COMM ARCOF
COMM SMOVL C00540 BC00540 V=400.0  +MOVJ EC00540
COMM SMOVL C00541 BC00541 V=1000.0  +MOVJ EC00541
COMM SFTOF3D
'Path W1887
SFTOF3D
SFTON3D P023
MOVJ C00542 BC00542 VJ=100.00  +MOVJ EC00542 VJ=100.00
SMOVL C00543 BC00543 V=400.0  +MOVJ EC00543
SMOVL C00544 BC00544 V=100.0 PL=0  +MOVJ EC00544
SREFP 1 C00545 BC00545  +REFP EC00545
SREFP 2 C00546 BC00546  +REFP EC00546
MACRO1 MJ#(0) ARGF9
ARCON
SMOVL C00547 BC00547 V=10.0  +MOVJ EC00547
ARCOF
SMOVL C00548 BC00548 V=400.0  +MOVJ EC00548
SMOVL C00549 BC00549 V=1000.0  +MOVJ EC00549
SFTOF3D
MOVJ C00550 BC00550 VJ=100.00  +MOVJ EC00550 VJ=100.00
MOVJ C00551 BC00551 VJ=100.00  +MOVJ EC00551 VJ=100.00
MOVJ C00552 BC00552 VJ=100.00  +MOVJ EC00552 VJ=100.00
'2
MOVJ C00553 BC00553 VJ=100.00  +MOVJ EC00553 VJ=100.00
MOVJ C00554 BC00554 VJ=100.00  +MOVJ EC00554 VJ=20.00
MOVJ C00555 BC00555 VJ=100.00  +MOVJ EC00555 VJ=100.00
'Path W1888
SFTOF3D
SFTON3D P021
MOVJ C00556 BC00556 VJ=15.00  +MOVJ EC00556 VJ=100.00
SMOVL C00557 BC00557 V=400.0  +MOVJ EC00557
SMOVL C00558 BC00558 V=133.3 PL=0  +MOVJ EC00558
SREFP 1 C00559 BC00559  +REFP EC00559
SREFP 2 C00560 BC00560  +REFP EC00560
MACRO1 MJ#(0) ARGF14
ARCON
SMOVL C00561 BC00561 V=10.0  +MOVJ EC00561
ARCOF
SMOVL C00562 BC00562 V=166.7  +MOVJ EC00562
SMOVL C00563 BC00563 V=166.7  +MOVJ EC00563
MACRO1 MJ#(0) ARGF14
SMOVL C00564 BC00564 V=133.3 PL=0  +MOVJ EC00564
ARCON
SMOVL C00565 BC00565 V=10.0  +MOVJ EC00565
ARCOF
SMOVL C00566 BC00566 V=400.0  +MOVJ EC00566
SFTOF3D
MOVJ C00567 BC00567 VJ=50.00  +MOVJ EC00567 VJ=20.00
MOVJ C00568 BC00568 VJ=100.00  +MOVJ EC00568 VJ=100.00
'Path W1889
SFTOF3D
SFTON3D P021
MOVJ C00569 BC00569 VJ=100.00  +MOVJ EC00569 VJ=100.00
MOVJ C00570 BC00570 VJ=100.00  +MOVJ EC00570 VJ=100.00
SMOVL C00571 BC00571 V=400.0  +MOVJ EC00571
SMOVL C00572 BC00572 V=133.3 PL=0  +MOVJ EC00572
SREFP 1 C00573 BC00573  +REFP EC00573
SREFP 2 C00574 BC00574  +REFP EC00574
MACRO1 MJ#(0) ARGF14
ARCON
SMOVL C00575 BC00575 V=10.0  +MOVJ EC00575
ARCOF
SMOVL C00576 BC00576 V=166.7  +MOVJ EC00576
SMOVL C00577 BC00577 V=166.7  +MOVJ EC00577
SMOVL C00578 BC00578 V=166.7 PL=0  +MOVJ EC00578
ARCON
SMOVL C00579 BC00579 V=10.0  +MOVJ EC00579
ARCOF
SMOVL C00580 BC00580 V=400.0  +MOVJ EC00580
SMOVL C00581 BC00581 V=1000.0  +MOVJ EC00581
SMOVL C00582 BC00582 V=1000.0  +MOVJ EC00582
SFTOF3D
MOVJ C00583 BC00583 VJ=100.00  +MOVJ EC00583 VJ=20.00
MOVJ C00584 BC00584 VJ=100.00  +MOVJ EC00584 VJ=100.00
MOVJ C00585 BC00585 VJ=100.00  +MOVJ EC00585 VJ=100.00
MOVJ C00586 BC00586 VJ=100.00  +MOVJ EC00586 VJ=100.00
MOVJ C00587 BC00587 VJ=100.00  +MOVJ EC00587 VJ=100.00
'3
'Path W1890
SFTOF3D
SFTON3D P023
MOVJ C00588 BC00588 VJ=100.00  +MOVJ EC00588 VJ=100.00
'BRAKUJACY ELEMENT
COMM SMOVL C00589 BC00589 V=400.0  +MOVJ EC00589
COMM SMOVL C00590 BC00590 V=100.0 PL=0  +MOVJ EC00590
COMM SREFP 1 C00591 BC00591  +REFP EC00591
COMM SREFP 2 C00592 BC00592  +REFP EC00592
COMM MACRO1 MJ#(0) ARGF0
COMM ARCON
COMM SMOVL C00593 BC00593 V=10.0  +MOVJ EC00593
COMM SMOVL C00594 BC00594 V=10.0  +MOVJ EC00594
COMM SMOVL C00595 BC00595 V=10.0  +MOVJ EC00595
COMM ARCOF
COMM SMOVL C00596 BC00596 V=400.0  +MOVJ EC00596
COMM SMOVL C00597 BC00597 V=1000.0  +MOVJ EC00597
SFTOF3D
'Path W1891
SFTOF3D
SFTON3D P023
MOVJ C00598 BC00598 VJ=100.00  +MOVJ EC00598 VJ=100.00
SMOVL C00599 BC00599 V=400.0  +MOVJ EC00599
SMOVL C00600 BC00600 V=133.3 PL=0  +MOVJ EC00600
SREFP 1 C00601 BC00601  +REFP EC00601
SREFP 2 C00602 BC00602  +REFP EC00602
MACRO1 MJ#(0) ARGF14
ARCON
SMOVL C00603 BC00603 V=11.7  +MOVJ EC00603
ARCOF
SMOVL C00604 BC00604 V=400.0  +MOVJ EC00604
SMOVL C00605 BC00605 V=1000.0  +MOVJ EC00605
SFTOF3D
MOVJ C00606 BC00606 VJ=100.00  +MOVJ EC00606 VJ=100.00
MOVJ C00607 BC00607 VJ=100.00  +MOVJ EC00607 VJ=20.00
MOVJ C00608 BC00608 VJ=100.00  +MOVJ EC00608 VJ=100.00
MOVJ C00609 BC00609 VJ=100.00  +MOVJ EC00609 VJ=20.00
MOVJ C00610 BC00610 VJ=100.00  +MOVJ EC00610 VJ=100.00
MOVJ C00611 BC00611 VJ=100.00  +MOVJ EC00611 VJ=100.00
'4
'Path W1892
SFTOF3D
SFTON3D P022
MOVJ C00612 BC00612 VJ=100.00  +MOVJ EC00612 VJ=20.00
SMOVL C00613 BC00613 V=400.0  +MOVJ EC00613
SMOVL C00614 BC00614 V=133.3 PL=0  +MOVJ EC00614
SREFP 1 C00615 BC00615  +REFP EC00615
SREFP 2 C00616 BC00616  +REFP EC00616
MACRO1 MJ#(0) ARGF14
ARCON
SMOVL C00617 BC00617 V=10.0  +MOVJ EC00617
ARCOF
SMOVL C00618 BC00618 V=400.0  +MOVJ EC00618
SMOVL C00619 BC00619 V=1000.0  +MOVJ EC00619
SFTOF3D
'Path W1893
SFTOF3D
SFTON3D P022
MOVJ C00620 BC00620 VJ=20.00  +MOVJ EC00620 VJ=100.00
SMOVL C00621 BC00621 V=400.0  +MOVJ EC00621
SMOVL C00622 BC00622 V=133.3 PL=0  +MOVJ EC00622
SREFP 1 C00623 BC00623  +REFP EC00623
SREFP 2 C00624 BC00624  +REFP EC00624
MACRO1 MJ#(0) ARGF14
ARCON
SMOVL C00625 BC00625 V=10.0  +MOVJ EC00625
ARCOF
SMOVL C00626 BC00626 V=400.0  +MOVJ EC00626
SMOVL C00627 BC00627 V=1000.0  +MOVJ EC00627
SFTOF3D
'6
'Path W1895
SFTOF3D
MOVJ C00628 BC00628 VJ=40.00  +MOVJ EC00628 VJ=100.00
SMOVL C00629 BC00629 V=400.0  +MOVJ EC00629
SFTON3D P022
SMOVL C00630 BC00630 V=133.3 PL=0  +MOVJ EC00630
SREFP 1 C00631 BC00631  +REFP EC00631
SREFP 2 C00632 BC00632  +REFP EC00632
MACRO1 MJ#(0) ARGF14
ARCON
SMOVL C00633 BC00633 V=11.7  +MOVJ EC00633
ARCOF
SMOVL C00634 BC00634 V=166.7  +MOVJ EC00634
SMOVL C00635 BC00635 V=166.7  +MOVJ EC00635
SMOVL C00636 BC00636 V=166.7 PL=0  +MOVJ EC00636
ARCON
SMOVL C00637 BC00637 V=11.7  +MOVJ EC00637
ARCOF
SMOVL C00638 BC00638 V=400.0  +MOVJ EC00638
SMOVL C00639 BC00639 V=1000.0  +MOVJ EC00639
SFTOF3D
MOVJ C00640 BC00640 VJ=100.00  +MOVJ EC00640 VJ=100.00
'Path W1896
SFTOF3D
SFTON3D P022
MOVJ C00641 BC00641 VJ=50.00  +MOVJ EC00641 VJ=100.00
SMOVL C00642 BC00642 V=400.0  +MOVJ EC00642
SMOVL C00643 BC00643 V=133.3 PL=0  +MOVJ EC00643
SREFP 1 C00644 BC00644  +REFP EC00644
SREFP 2 C00645 BC00645  +REFP EC00645
MACRO1 MJ#(0) ARGF14
ARCON
SMOVL C00646 BC00646 V=12.5  +MOVJ EC00646
ARCOF
SMOVL C00647 BC00647 V=400.0  +MOVJ EC00647
SMOVL C00648 BC00648 V=1000.0  +MOVJ EC00648
SFTOF3D
'7
'Path W1897
SFTOF3D
SFTON3D P022
MOVJ C00649 BC00649 VJ=100.00  +MOVJ EC00649 VJ=100.00
SMOVL C00650 BC00650 V=400.0  +MOVJ EC00650
SMOVL C00651 BC00651 V=133.3 PL=0  +MOVJ EC00651
SREFP 1 C00652 BC00652  +REFP EC00652
SREFP 2 C00653 BC00653  +REFP EC00653
MACRO1 MJ#(0) ARGF14
ARCON
SMOVL C00654 BC00654 V=12.5  +MOVJ EC00654
ARCOF
SMOVL C00655 BC00655 V=400.0  +MOVJ EC00655
SMOVL C00656 BC00656 V=1000.0  +MOVJ EC00656
SMOVL C00657 BC00657 V=1000.0  +MOVJ EC00657
SFTOF3D
MOVJ C00658 BC00658 VJ=100.00  +MOVJ EC00658 VJ=100.00
'Path W1898
SFTOF3D
SFTON3D P022
MOVJ C00659 BC00659 VJ=100.00  +MOVJ EC00659 VJ=100.00
SMOVL C00660 BC00660 V=400.0  +MOVJ EC00660
SMOVL C00661 BC00661 V=133.3 PL=0  +MOVJ EC00661
SREFP 1 C00662 BC00662  +REFP EC00662
SREFP 2 C00663 BC00663  +REFP EC00663
MACRO1 MJ#(0) ARGF14
ARCON
SMOVL C00664 BC00664 V=12.5  +MOVJ EC00664
ARCOF
SFTOF3D
SMOVL C00665 BC00665 V=400.0  +MOVJ EC00665
SMOVL C00666 BC00666 V=1000.0  +MOVJ EC00666
MOVJ C00667 BC00667 VJ=100.00  +MOVJ EC00667 VJ=20.00
MOVJ C00668 BC00668 VJ=100.00  +MOVJ EC00668 VJ=100.00
SFTOF3D
END
